// TIA Portal V18 export
FUNCTION "ST10_Auto" : Void   // FC1003, LAD
{ S7_Optimized_Access := 'FALSE' }
// stored: AutoNumber false, SetENOAutomatically false
   VAR_INPUT
      iSysMode : "RCS_SysComInterface_V1";
   END_VAR
   VAR_TEMP
      i : Int;
      tBool : Bool;
      FlankWord : Int;
   END_VAR
   VAR_TEMP   // added for the SCL form of the ladder/FBD networks
      _w1 : Bool;
      _w2 : Bool;
      _w3 : Bool;
      _w4 : Bool;
      _w5 : Bool;
      _w6 : Bool;
   END_VAR
BEGIN

REGION Network 1
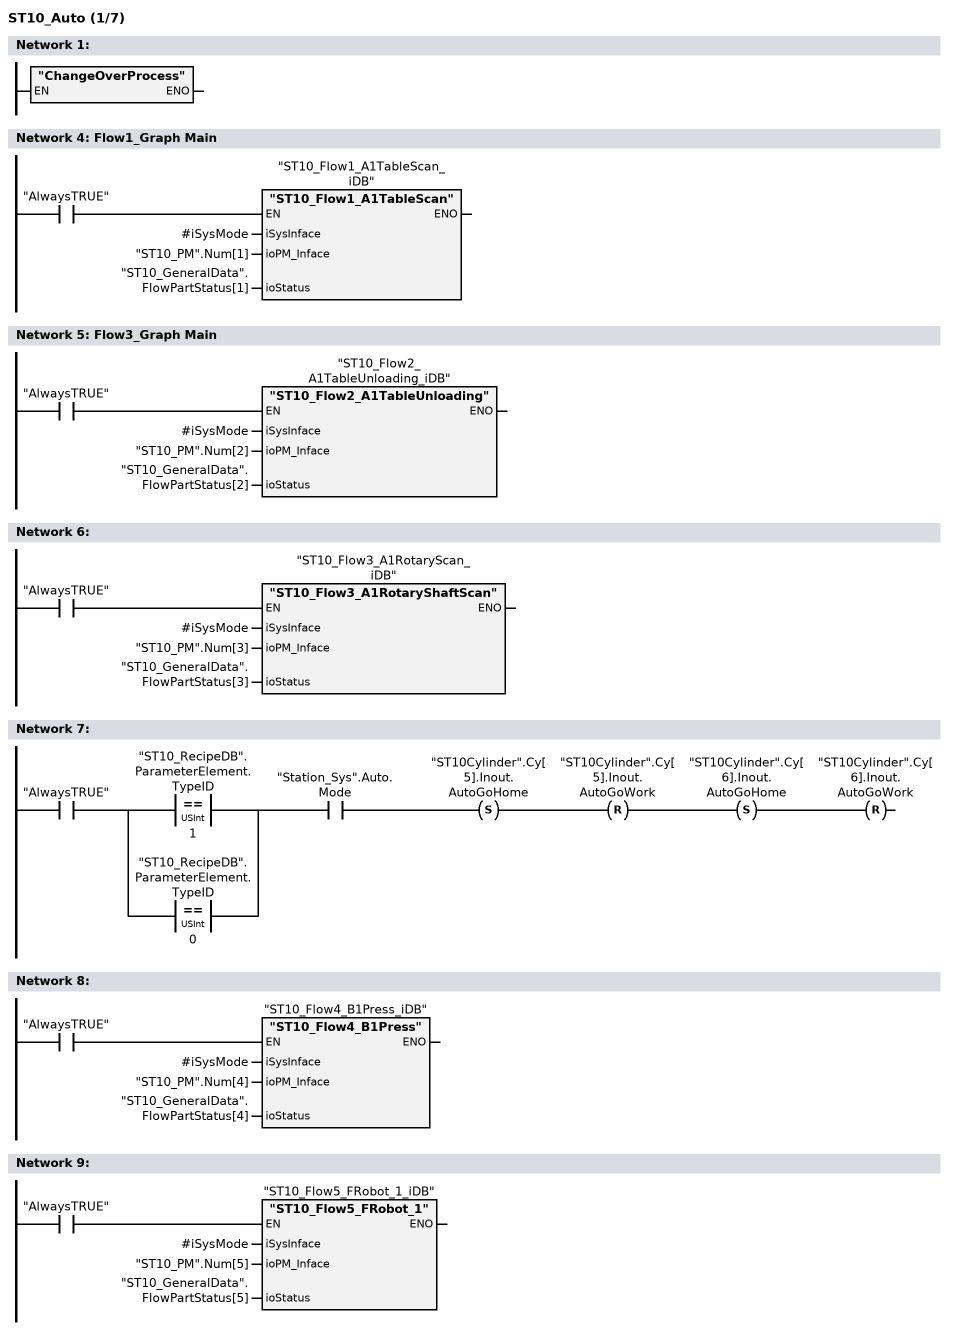
   RUNG wire#powerrail
      "ChangeOverProcess"()
   END_RUNG
   // the same network as SCL:
   "ChangeOverProcess"();
END_REGION

NETWORK
TITLE = AutoMain//自动
//Autorunning is not allowed in manual mode
      A     "Station_Sys".Manual.Mode;
      R     "Station_Sys".Auto.Running;
//one cycle interface
      A     "Station_Sys".Cmd.OneCycle;
      =     "ST10_PM".Num[1].TriggerOneCycle;
      =     "ST10_PM".Num[2].TriggerOneCycle;
      =     "ST10_PM".Num[3].TriggerOneCycle;
      =     "ST10_PM".Num[4].TriggerOneCycle;
      =     "ST10_PM".Num[5].TriggerOneCycle;
      =     "ST10_PM".Num[6].TriggerOneCycle;
      =     "ST10_PM".Num[7].TriggerOneCycle;
      =     "ST10_PM".Num[8].TriggerOneCycle;
      =     "ST10_PM".Num[11].TriggerOneCycle;
      =     "ST10_PM".Num[12].TriggerOneCycle;
      =     "ST10_PM".Num[14].TriggerOneCycle;
      =     "ST10_PM".Num[15].TriggerOneCycle;
      =     "ST10_PM".Num[16].TriggerOneCycle;
      =     "ST10_PM".Num[21].TriggerOneCycle;
      =     "ST10_PM".Num[22].TriggerOneCycle;
      =     "ST10_PM".Num[23].TriggerOneCycle;
      =     "ST10_PM".Num[24].TriggerOneCycle;


NETWORK
TITLE = InitialStatus-初始化状态
//Initilizing
      O     "ST10_PM".Num[1].InitialRun;
      O     "ST10_PM".Num[2].InitialRun;
      O     "ST10_PM".Num[3].InitialRun;
      O     "ST10_PM".Num[4].InitialRun;
      O     "ST10_PM".Num[5].InitialRun;
      O     "ST10_PM".Num[6].InitialRun;
      O     "ST10_PM".Num[7].InitialRun;
      O     "ST10_PM".Num[8].InitialRun;
      O     "ST10_PM".Num[11].InitialRun;
      O     "ST10_PM".Num[12].InitialRun;
      O     "ST10_PM".Num[14].InitialRun;
      O     "ST10_PM".Num[15].InitialRun;
      O     "ST10_PM".Num[21].InitialRun;
      O     "ST10_PM".Num[22].InitialRun;
      O     "ST10_PM".Num[23].InitialRun;
      O     "ST10_PM".Num[24].InitialRun;
      =     "Station_Sys".Initial.Running;
//Initilize ok

      A     "ST10_PM".Num[1].InitialOK;
      A     "ST10_PM".Num[2].InitialOK;
      A     "ST10_PM".Num[3].InitialOK;
      A     "ST10_PM".Num[4].InitialOK;
      A     "ST10_PM".Num[5].InitialOK;
      A     "ST10_PM".Num[6].InitialOK;
      A     "ST10_PM".Num[7].InitialOK;
      A     "ST10_PM".Num[8].InitialOK;
      A     "ST10_PM".Num[11].InitialOK;
      A     "ST10_PM".Num[12].InitialOK;
      A     "ST10_PM".Num[14].InitialOK;
      A     "ST10_PM".Num[15].InitialOK;

      A     "ST10_PM".Num[21].InitialOK;
      A     "ST10_PM".Num[22].InitialOK;
      A     "ST10_PM".Num[23].InitialOK;
      A     "ST10_PM".Num[24].InitialOK;
      =     "Station_Sys".Initial.OK;

//Auto running
      A     "Station_Sys".Auto.Mode;
      A(;
      O     "ST10_PM".Num[1].Running;
      O     "ST10_PM".Num[2].Running;
      O     "ST10_PM".Num[3].Running;
      O     "ST10_PM".Num[4].Running;
      O     "ST10_PM".Num[5].Running;
      O     "ST10_PM".Num[6].Running;
      O     "ST10_PM".Num[7].Running;
      O     "ST10_PM".Num[8].Running;
      O     "ST10_PM".Num[11].Running;
      O     "ST10_PM".Num[12].Running;
      O     "ST10_PM".Num[14].Running;
      O     "ST10_PM".Num[15].Running;

      O     "ST10_PM".Num[21].Running;
      O     "ST10_PM".Num[22].Running;
      O     "ST10_PM".Num[23].Running;
      O     "ST10_PM".Num[24].Running;
      );
// AN    "Station_Sys".Auto.AllRun
      =     "Station_Sys".Auto.Running;
//All run
      A     "ST10_PM".Num[1].Running;
      A     "ST10_PM".Num[2].Running;
      A     "ST10_PM".Num[3].Running;
      A     "ST10_PM".Num[4].Running;
      A     "ST10_PM".Num[5].Running;
      A     "ST10_PM".Num[6].Running;
      A     "ST10_PM".Num[7].Running;
      A     "ST10_PM".Num[8].Running;
      A     "ST10_PM".Num[11].Running;
      A     "ST10_PM".Num[12].Running;
      A     "ST10_PM".Num[14].Running;
      A     "ST10_PM".Num[15].Running;

      A     "ST10_PM".Num[21].Running;
      A     "ST10_PM".Num[22].Running;
      A     "ST10_PM".Num[23].Running;
      A     "ST10_PM".Num[24].Running;
      =     "Station_Sys".Auto.AllRun;




REGION Network 4: Flow1_Graph Main
   RUNG wire#powerrail
      Contact( "AlwaysTRUE" )
      "ST10_Flow1_A1TableScan_iDB"(iSysInface := #iSysMode, ioPM_Inface := "ST10_PM".Num[1], ioStatus := "ST10_GeneralData".FlowPartStatus[1])
   END_RUNG
   // the same network as SCL:
   IF "AlwaysTRUE" THEN
       "ST10_Flow1_A1TableScan_iDB"(iSysInface := #iSysMode,   // "ST10_Flow1_A1TableScan"
                               ioPM_Inface := "ST10_PM".Num[1],
                               ioStatus := "ST10_GeneralData".FlowPartStatus[1]);
   END_IF;
END_REGION

REGION Network 5: Flow3_Graph Main
   RUNG wire#powerrail
      Contact( "AlwaysTRUE" )
      "ST10_Flow2_A1TableUnloading_iDB"(iSysInface := #iSysMode, ioPM_Inface := "ST10_PM".Num[2], ioStatus := "ST10_GeneralData".FlowPartStatus[2])
   END_RUNG
   // the same network as SCL:
   IF "AlwaysTRUE" THEN
       "ST10_Flow2_A1TableUnloading_iDB"(iSysInface := #iSysMode,   // "ST10_Flow2_A1TableUnloading"
                               ioPM_Inface := "ST10_PM".Num[2],
                               ioStatus := "ST10_GeneralData".FlowPartStatus[2]);
   END_IF;
END_REGION

REGION Network 6
   RUNG wire#powerrail
      Contact( "AlwaysTRUE" )
      "ST10_Flow3_A1RotaryScan_iDB"(iSysInface := #iSysMode, ioPM_Inface := "ST10_PM".Num[3], ioStatus := "ST10_GeneralData".FlowPartStatus[3])
   END_RUNG
   // the same network as SCL:
   IF "AlwaysTRUE" THEN
       "ST10_Flow3_A1RotaryScan_iDB"(iSysInface := #iSysMode,   // "ST10_Flow3_A1RotaryShaftScan"
                               ioPM_Inface := "ST10_PM".Num[3],
                               ioStatus := "ST10_GeneralData".FlowPartStatus[3]);
   END_IF;
END_REGION

REGION Network 7
   RUNG wire#powerrail
      Contact( "AlwaysTRUE" )
      wire#w1
      { S7_Templates := "SrcType := USInt" } EQ_Contact(in1 := "ST10_RecipeDB".ParameterElement.TypeID, in2 := 1)
      wire#w2
      Contact( "Station_Sys".Auto.Mode )
      S_Coil( "ST10Cylinder".Cy[5].Inout.AutoGoHome )
      R_Coil( "ST10Cylinder".Cy[5].Inout.AutoGoWork )
      S_Coil( "ST10Cylinder".Cy[6].Inout.AutoGoHome )
      R_Coil( "ST10Cylinder".Cy[6].Inout.AutoGoWork )
   END_RUNG
   RUNG wire#w1
      { S7_Templates := "SrcType := USInt" } EQ_Contact(in1 := "ST10_RecipeDB".ParameterElement.TypeID, in2 := 0)
   END_RUNG wire#w2
   // the same network as SCL:
   IF "AlwaysTRUE" AND (("ST10_RecipeDB".ParameterElement.TypeID = 1) OR ("ST10_RecipeDB".ParameterElement.TypeID = 0)) AND "Station_Sys".Auto.Mode THEN
       "ST10Cylinder".Cy[5].Inout.AutoGoHome := TRUE;
       "ST10Cylinder".Cy[5].Inout.AutoGoWork := FALSE;
       "ST10Cylinder".Cy[6].Inout.AutoGoHome := TRUE;
       "ST10Cylinder".Cy[6].Inout.AutoGoWork := FALSE;
   END_IF;
END_REGION

REGION Network 8
   RUNG wire#powerrail
      Contact( "AlwaysTRUE" )
      "ST10_Flow4_B1Press_iDB"(iSysInface := #iSysMode, ioPM_Inface := "ST10_PM".Num[4], ioStatus := "ST10_GeneralData".FlowPartStatus[4])
   END_RUNG
   // the same network as SCL:
   IF "AlwaysTRUE" THEN
       "ST10_Flow4_B1Press_iDB"(iSysInface := #iSysMode,   // "ST10_Flow4_B1Press"
                               ioPM_Inface := "ST10_PM".Num[4],
                               ioStatus := "ST10_GeneralData".FlowPartStatus[4]);
   END_IF;
END_REGION

REGION Network 9
   RUNG wire#powerrail
      Contact( "AlwaysTRUE" )
      "ST10_Flow5_FRobot_1_iDB"(iSysInface := #iSysMode, ioPM_Inface := "ST10_PM".Num[5], ioStatus := "ST10_GeneralData".FlowPartStatus[5])
   END_RUNG
   // the same network as SCL:
   IF "AlwaysTRUE" THEN
       "ST10_Flow5_FRobot_1_iDB"(iSysInface := #iSysMode,   // "ST10_Flow5_FRobot_1"
                               ioPM_Inface := "ST10_PM".Num[5],
                               ioStatus := "ST10_GeneralData".FlowPartStatus[5]);
   END_IF;
END_REGION

REGION Network 10
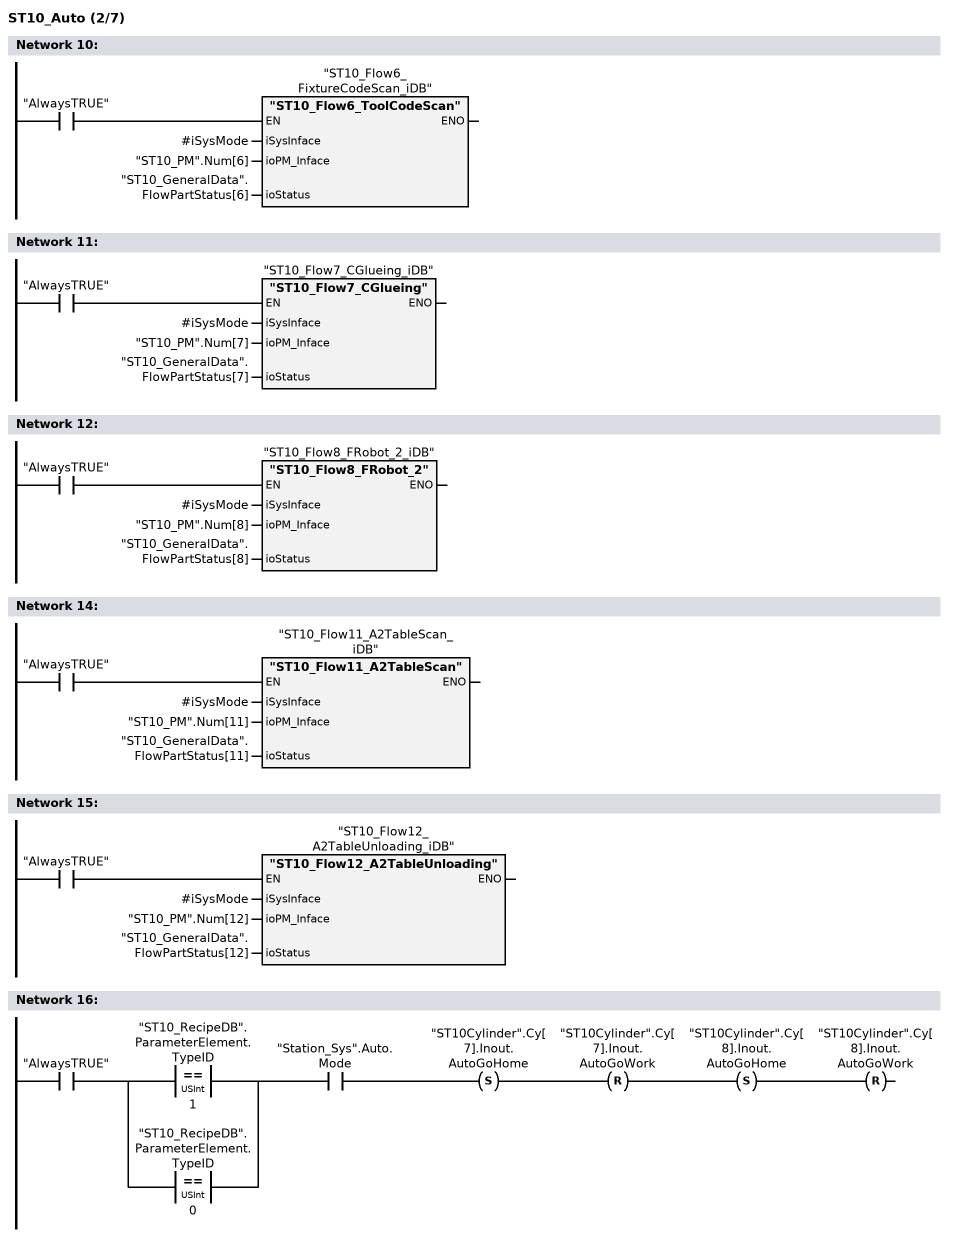
   RUNG wire#powerrail
      Contact( "AlwaysTRUE" )
      "ST10_Flow6_FixtureCodeScan_iDB"(iSysInface := #iSysMode, ioPM_Inface := "ST10_PM".Num[6], ioStatus := "ST10_GeneralData".FlowPartStatus[6])
   END_RUNG
   // the same network as SCL:
   IF "AlwaysTRUE" THEN
       "ST10_Flow6_FixtureCodeScan_iDB"(iSysInface := #iSysMode,   // "ST10_Flow6_ToolCodeScan"
                               ioPM_Inface := "ST10_PM".Num[6],
                               ioStatus := "ST10_GeneralData".FlowPartStatus[6]);
   END_IF;
END_REGION

REGION Network 11
   RUNG wire#powerrail
      Contact( "AlwaysTRUE" )
      "ST10_Flow7_CGlueing_iDB"(iSysInface := #iSysMode, ioPM_Inface := "ST10_PM".Num[7], ioStatus := "ST10_GeneralData".FlowPartStatus[7])
   END_RUNG
   // the same network as SCL:
   IF "AlwaysTRUE" THEN
       "ST10_Flow7_CGlueing_iDB"(iSysInface := #iSysMode,   // "ST10_Flow7_CGlueing"
                               ioPM_Inface := "ST10_PM".Num[7],
                               ioStatus := "ST10_GeneralData".FlowPartStatus[7]);
   END_IF;
END_REGION

REGION Network 12
   RUNG wire#powerrail
      Contact( "AlwaysTRUE" )
      "ST10_Flow8_FRobot_2_iDB"(iSysInface := #iSysMode, ioPM_Inface := "ST10_PM".Num[8], ioStatus := "ST10_GeneralData".FlowPartStatus[8])
   END_RUNG
   // the same network as SCL:
   IF "AlwaysTRUE" THEN
       "ST10_Flow8_FRobot_2_iDB"(iSysInface := #iSysMode,   // "ST10_Flow8_FRobot_2"
                               ioPM_Inface := "ST10_PM".Num[8],
                               ioStatus := "ST10_GeneralData".FlowPartStatus[8]);
   END_IF;
END_REGION

REGION Network 14
   RUNG wire#powerrail
      Contact( "AlwaysTRUE" )
      "ST10_Flow11_A2TableScan_iDB"(iSysInface := #iSysMode, ioPM_Inface := "ST10_PM".Num[11], ioStatus := "ST10_GeneralData".FlowPartStatus[11])
   END_RUNG
   // the same network as SCL:
   IF "AlwaysTRUE" THEN
       "ST10_Flow11_A2TableScan_iDB"(iSysInface := #iSysMode,   // "ST10_Flow11_A2TableScan"
                               ioPM_Inface := "ST10_PM".Num[11],
                               ioStatus := "ST10_GeneralData".FlowPartStatus[11]);
   END_IF;
END_REGION

REGION Network 15
   RUNG wire#powerrail
      Contact( "AlwaysTRUE" )
      "ST10_Flow12_A2TableUnloading_iDB"(iSysInface := #iSysMode, ioPM_Inface := "ST10_PM".Num[12], ioStatus := "ST10_GeneralData".FlowPartStatus[12])
   END_RUNG
   // the same network as SCL:
   IF "AlwaysTRUE" THEN
       "ST10_Flow12_A2TableUnloading_iDB"(iSysInface := #iSysMode,   // "ST10_Flow12_A2TableUnloading"
                               ioPM_Inface := "ST10_PM".Num[12],
                               ioStatus := "ST10_GeneralData".FlowPartStatus[12]);
   END_IF;
END_REGION

REGION Network 16
   RUNG wire#powerrail
      Contact( "AlwaysTRUE" )
      wire#w1
      { S7_Templates := "SrcType := USInt" } EQ_Contact(in1 := "ST10_RecipeDB".ParameterElement.TypeID, in2 := 1)
      wire#w2
      Contact( "Station_Sys".Auto.Mode )
      S_Coil( "ST10Cylinder".Cy[7].Inout.AutoGoHome )
      R_Coil( "ST10Cylinder".Cy[7].Inout.AutoGoWork )
      S_Coil( "ST10Cylinder".Cy[8].Inout.AutoGoHome )
      R_Coil( "ST10Cylinder".Cy[8].Inout.AutoGoWork )
   END_RUNG
   RUNG wire#w1
      { S7_Templates := "SrcType := USInt" } EQ_Contact(in1 := "ST10_RecipeDB".ParameterElement.TypeID, in2 := 0)
   END_RUNG wire#w2
   // the same network as SCL:
   IF "AlwaysTRUE" AND (("ST10_RecipeDB".ParameterElement.TypeID = 1) OR ("ST10_RecipeDB".ParameterElement.TypeID = 0)) AND "Station_Sys".Auto.Mode THEN
       "ST10Cylinder".Cy[7].Inout.AutoGoHome := TRUE;
       "ST10Cylinder".Cy[7].Inout.AutoGoWork := FALSE;
       "ST10Cylinder".Cy[8].Inout.AutoGoHome := TRUE;
       "ST10Cylinder".Cy[8].Inout.AutoGoWork := FALSE;
   END_IF;
END_REGION

REGION Network 17
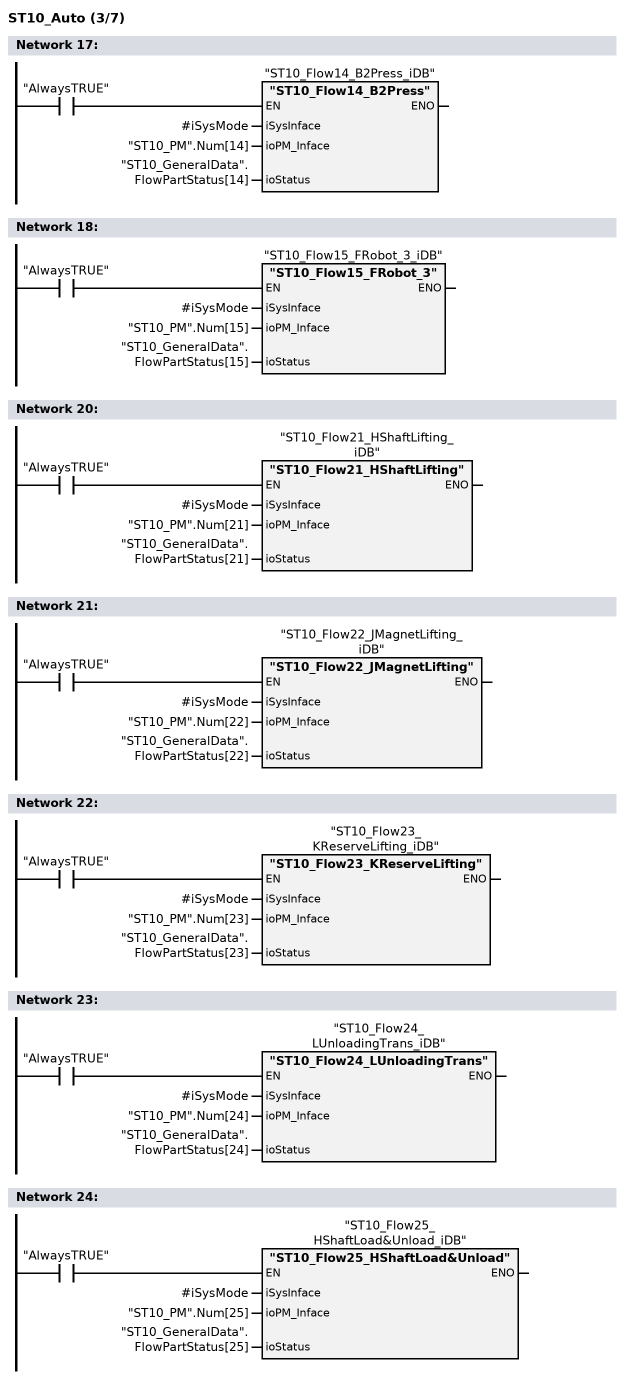
   RUNG wire#powerrail
      Contact( "AlwaysTRUE" )
      "ST10_Flow14_B2Press_iDB"(iSysInface := #iSysMode, ioPM_Inface := "ST10_PM".Num[14], ioStatus := "ST10_GeneralData".FlowPartStatus[14])
   END_RUNG
   // the same network as SCL:
   IF "AlwaysTRUE" THEN
       "ST10_Flow14_B2Press_iDB"(iSysInface := #iSysMode,   // "ST10_Flow14_B2Press"
                               ioPM_Inface := "ST10_PM".Num[14],
                               ioStatus := "ST10_GeneralData".FlowPartStatus[14]);
   END_IF;
END_REGION

REGION Network 18
   RUNG wire#powerrail
      Contact( "AlwaysTRUE" )
      "ST10_Flow15_FRobot_3_iDB"(iSysInface := #iSysMode, ioPM_Inface := "ST10_PM".Num[15], ioStatus := "ST10_GeneralData".FlowPartStatus[15])
   END_RUNG
   // the same network as SCL:
   IF "AlwaysTRUE" THEN
       "ST10_Flow15_FRobot_3_iDB"(iSysInface := #iSysMode,   // "ST10_Flow15_FRobot_3"
                               ioPM_Inface := "ST10_PM".Num[15],
                               ioStatus := "ST10_GeneralData".FlowPartStatus[15]);
   END_IF;
END_REGION

REGION Network 20
   RUNG wire#powerrail
      Contact( "AlwaysTRUE" )
      "ST10_Flow21_HShaftLifting_iDB"(iSysInface := #iSysMode, ioPM_Inface := "ST10_PM".Num[21], ioStatus := "ST10_GeneralData".FlowPartStatus[21])
   END_RUNG
   // the same network as SCL:
   IF "AlwaysTRUE" THEN
       "ST10_Flow21_HShaftLifting_iDB"(iSysInface := #iSysMode,   // "ST10_Flow21_HShaftLifting"
                               ioPM_Inface := "ST10_PM".Num[21],
                               ioStatus := "ST10_GeneralData".FlowPartStatus[21]);
   END_IF;
END_REGION

REGION Network 21
   RUNG wire#powerrail
      Contact( "AlwaysTRUE" )
      "ST10_Flow22_JMagnetLifting_iDB"(iSysInface := #iSysMode, ioPM_Inface := "ST10_PM".Num[22], ioStatus := "ST10_GeneralData".FlowPartStatus[22])
   END_RUNG
   // the same network as SCL:
   IF "AlwaysTRUE" THEN
       "ST10_Flow22_JMagnetLifting_iDB"(iSysInface := #iSysMode,   // "ST10_Flow22_JMagnetLifting"
                               ioPM_Inface := "ST10_PM".Num[22],
                               ioStatus := "ST10_GeneralData".FlowPartStatus[22]);
   END_IF;
END_REGION

REGION Network 22
   RUNG wire#powerrail
      Contact( "AlwaysTRUE" )
      "ST10_Flow23_KReserveLifting_iDB"(iSysInface := #iSysMode, ioPM_Inface := "ST10_PM".Num[23], ioStatus := "ST10_GeneralData".FlowPartStatus[23])
   END_RUNG
   // the same network as SCL:
   IF "AlwaysTRUE" THEN
       "ST10_Flow23_KReserveLifting_iDB"(iSysInface := #iSysMode,   // "ST10_Flow23_KReserveLifting"
                               ioPM_Inface := "ST10_PM".Num[23],
                               ioStatus := "ST10_GeneralData".FlowPartStatus[23]);
   END_IF;
END_REGION

REGION Network 23
   RUNG wire#powerrail
      Contact( "AlwaysTRUE" )
      "ST10_Flow24_LUnloadingTrans_iDB"(iSysInface := #iSysMode, ioPM_Inface := "ST10_PM".Num[24], ioStatus := "ST10_GeneralData".FlowPartStatus[24])
   END_RUNG
   // the same network as SCL:
   IF "AlwaysTRUE" THEN
       "ST10_Flow24_LUnloadingTrans_iDB"(iSysInface := #iSysMode,   // "ST10_Flow24_LUnloadingTrans"
                               ioPM_Inface := "ST10_PM".Num[24],
                               ioStatus := "ST10_GeneralData".FlowPartStatus[24]);
   END_IF;
END_REGION

REGION Network 24
   RUNG wire#powerrail
      Contact( "AlwaysTRUE" )
      "ST10_Flow25_HShaftLoad&Unload_iDB"(iSysInface := #iSysMode, ioPM_Inface := "ST10_PM".Num[25], ioStatus := "ST10_GeneralData".FlowPartStatus[25])
   END_RUNG
   // the same network as SCL:
   IF "AlwaysTRUE" THEN
       "ST10_Flow25_HShaftLoad&Unload_iDB"(iSysInface := #iSysMode,   // "ST10_Flow25_HShaftLoad&Unload"
                               ioPM_Inface := "ST10_PM".Num[25],
                               ioStatus := "ST10_GeneralData".FlowPartStatus[25]);
   END_IF;
END_REGION

REGION Network 25
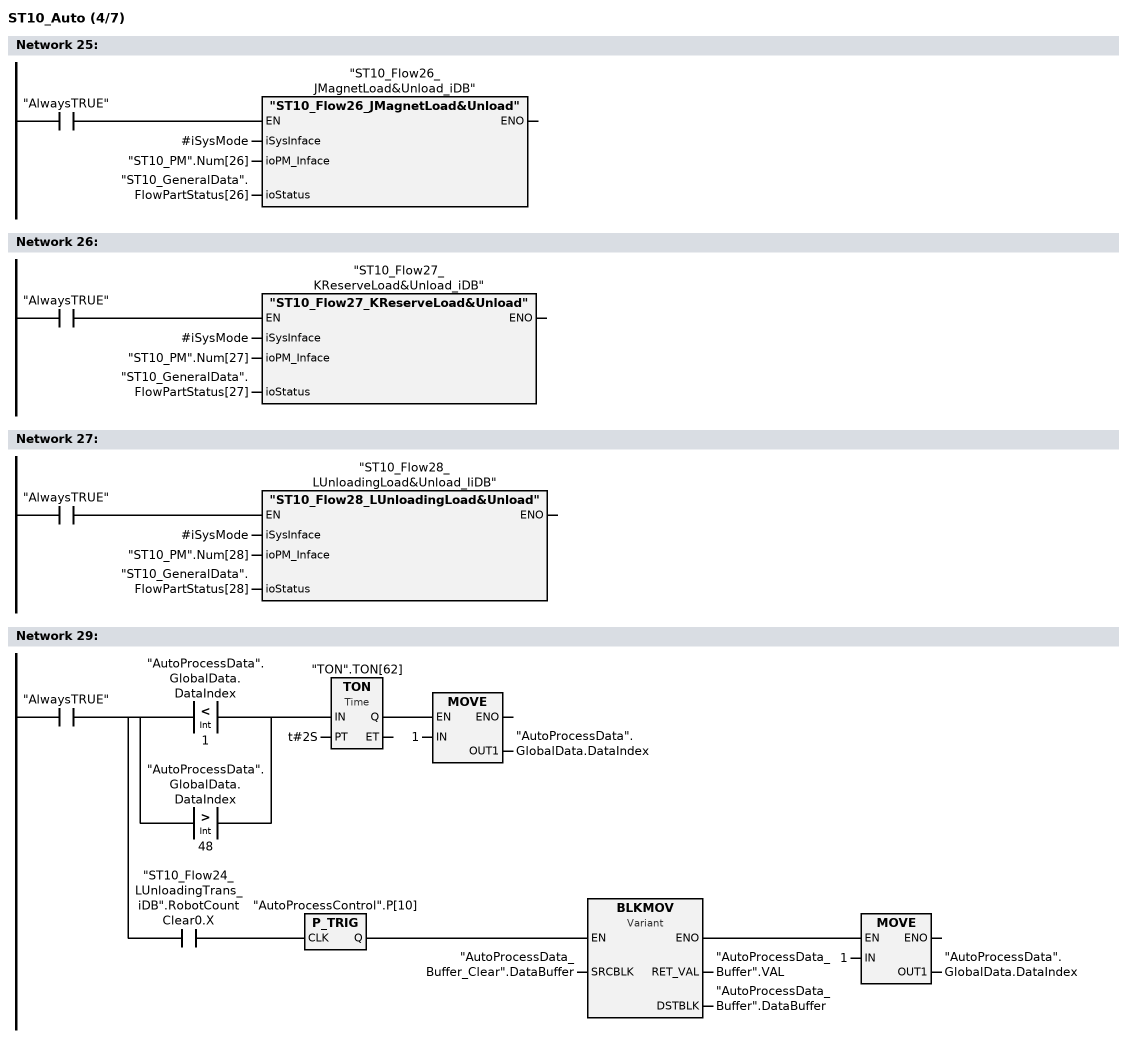
   RUNG wire#powerrail
      Contact( "AlwaysTRUE" )
      "ST10_Flow26_JMagnetLoad&Unload_iDB"(iSysInface := #iSysMode, ioPM_Inface := "ST10_PM".Num[26], ioStatus := "ST10_GeneralData".FlowPartStatus[26])
   END_RUNG
   // the same network as SCL:
   IF "AlwaysTRUE" THEN
       "ST10_Flow26_JMagnetLoad&Unload_iDB"(iSysInface := #iSysMode,   // "ST10_Flow26_JMagnetLoad&Unload"
                               ioPM_Inface := "ST10_PM".Num[26],
                               ioStatus := "ST10_GeneralData".FlowPartStatus[26]);
   END_IF;
END_REGION

REGION Network 26
   RUNG wire#powerrail
      Contact( "AlwaysTRUE" )
      "ST10_Flow27_KReserveLoad&Unload_iDB"(iSysInface := #iSysMode, ioPM_Inface := "ST10_PM".Num[27], ioStatus := "ST10_GeneralData".FlowPartStatus[27])
   END_RUNG
   // the same network as SCL:
   IF "AlwaysTRUE" THEN
       "ST10_Flow27_KReserveLoad&Unload_iDB"(iSysInface := #iSysMode,   // "ST10_Flow27_KReserveLoad&Unload"
                               ioPM_Inface := "ST10_PM".Num[27],
                               ioStatus := "ST10_GeneralData".FlowPartStatus[27]);
   END_IF;
END_REGION

REGION Network 27
   RUNG wire#powerrail
      Contact( "AlwaysTRUE" )
      "ST10_Flow28_LUnloadingLoad&Unload_IiDB"(iSysInface := #iSysMode, ioPM_Inface := "ST10_PM".Num[28], ioStatus := "ST10_GeneralData".FlowPartStatus[28])
   END_RUNG
   // the same network as SCL:
   IF "AlwaysTRUE" THEN
       "ST10_Flow28_LUnloadingLoad&Unload_IiDB"(iSysInface := #iSysMode,   // "ST10_Flow28_LUnloadingLoad&Unload"
                               ioPM_Inface := "ST10_PM".Num[28],
                               ioStatus := "ST10_GeneralData".FlowPartStatus[28]);
   END_IF;
END_REGION

REGION Network 29
   RUNG wire#powerrail
      Contact( "AlwaysTRUE" )
      wire#w1
      { S7_Templates := "SrcType := Int" } LT_Contact(in1 := "AutoProcessData".GlobalData.DataIndex, in2 := 1)
      wire#w2
      { S7_Templates := "time_type := Time" } "TON".TON[62].TON(pt := t#2S, et =>)
      Move(in := 1, out1 => "AutoProcessData".GlobalData.DataIndex)
   END_RUNG
   RUNG wire#w1
      { S7_Templates := "SrcType := Int" } GT_Contact(in1 := "AutoProcessData".GlobalData.DataIndex, in2 := 48)
   END_RUNG wire#w2
   RUNG wire#w1
      Contact( "ST10_Flow24_LUnloadingTrans_iDB".RobotCountClear0.X )
      P_Trig( "AutoProcessControl".P[10] )
      { S7_Templates := "blk_type := Variant" } BLKMOV(SRCBLK := "AutoProcessData_Buffer_Clear".DataBuffer, RET_VAL => "AutoProcessData_Buffer".VAL, DSTBLK => "AutoProcessData_Buffer".DataBuffer)
      Move(in := 1, out1 => "AutoProcessData".GlobalData.DataIndex)
   END_RUNG
   // the same network as SCL:
   "TON".TON[62].TON(IN := "AlwaysTRUE" AND (("AutoProcessData".GlobalData.DataIndex < 1) OR ("AutoProcessData".GlobalData.DataIndex > 48)),
                     PT := t#2S);
   IF "TON".TON[62].Q THEN "AutoProcessData".GlobalData.DataIndex := 1; END_IF;
   #_w1 := "AlwaysTRUE" AND "ST10_Flow24_LUnloadingTrans_iDB".RobotCountClear0.X;
   #_w2 := #_w1 AND NOT "AutoProcessControl".P[10];   // rising edge
   "AutoProcessControl".P[10] := #_w1;
   "AutoProcessData_Buffer".VAL := BLKMOV(EN := #_w2,
                           SRCBLK := "AutoProcessData_Buffer_Clear".DataBuffer,
                           DSTBLK => "AutoProcessData_Buffer".DataBuffer,
                           ENO => #_w3);
   IF #_w3 THEN "AutoProcessData".GlobalData.DataIndex := 1; END_IF;
END_REGION

REGION Network 30
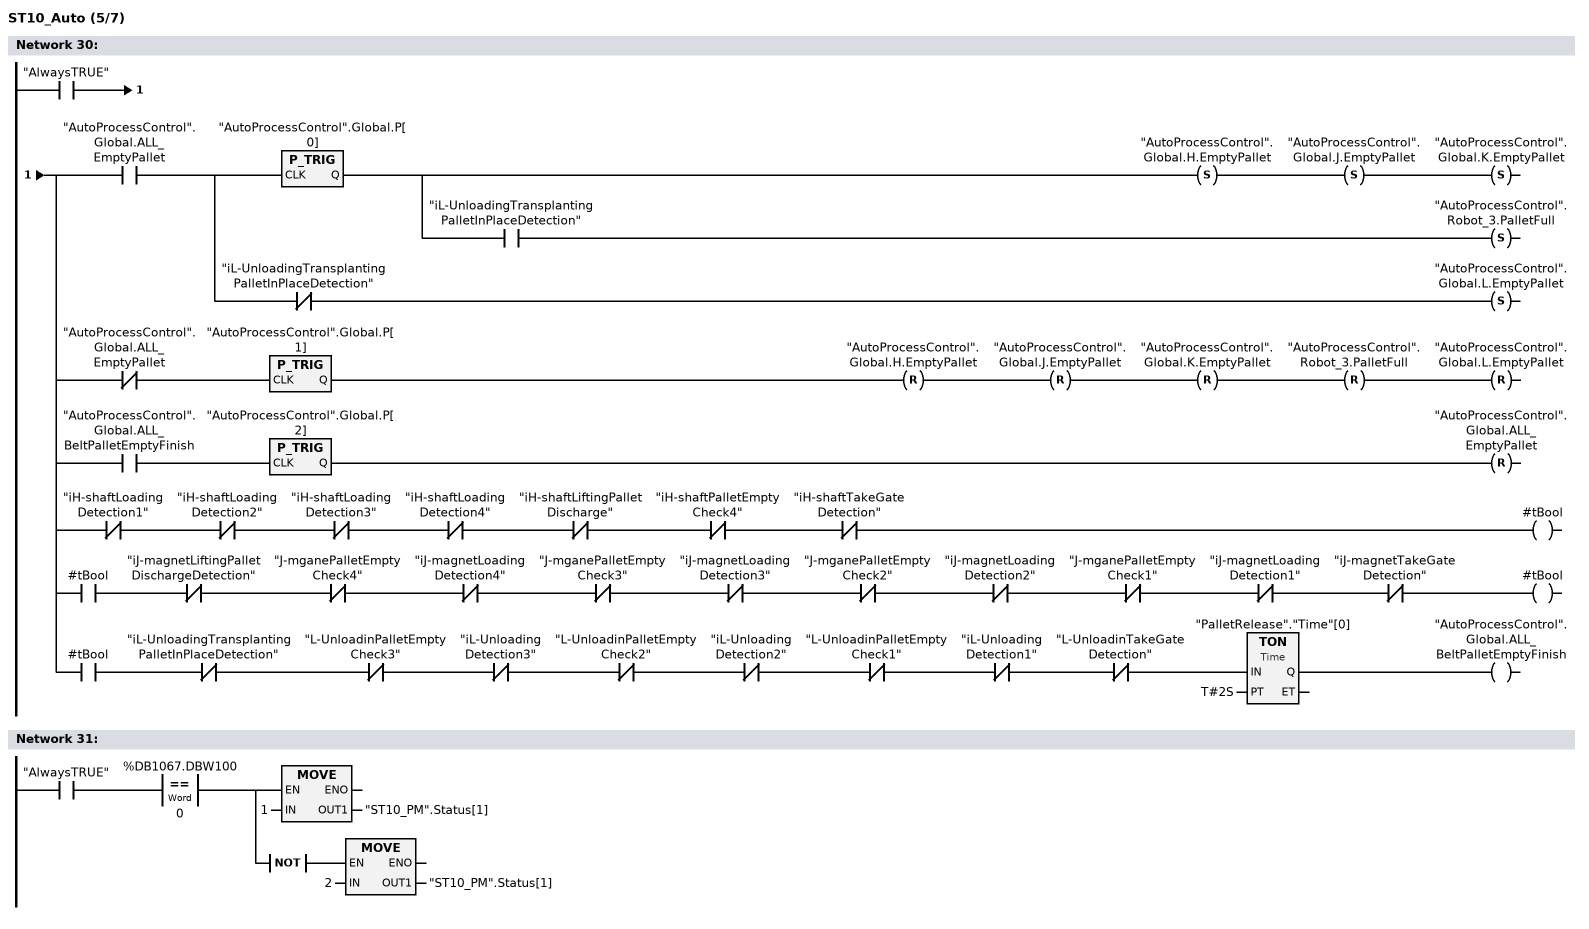
   RUNG wire#powerrail
      Contact( "AlwaysTRUE" )
      wire#w1
      Contact( "AutoProcessControl".Global.ALL_EmptyPallet )
      wire#w2
      P_Trig( "AutoProcessControl".Global.P[0] )
      wire#w3
      S_Coil( "AutoProcessControl".Global.H.EmptyPallet )
      S_Coil( "AutoProcessControl".Global.J.EmptyPallet )
      S_Coil( "AutoProcessControl".Global.K.EmptyPallet )
   END_RUNG
   RUNG wire#w3
      Contact( "iL-UnloadingTransplantingPalletInPlaceDetection" )
      S_Coil( "AutoProcessControl".Robot_3.PalletFull )
   END_RUNG
   RUNG wire#w2
      I_Contact( "iL-UnloadingTransplantingPalletInPlaceDetection" )
      S_Coil( "AutoProcessControl".Global.L.EmptyPallet )
   END_RUNG
   RUNG wire#w1
      I_Contact( "AutoProcessControl".Global.ALL_EmptyPallet )
      P_Trig( "AutoProcessControl".Global.P[1] )
      R_Coil( "AutoProcessControl".Global.H.EmptyPallet )
      R_Coil( "AutoProcessControl".Global.J.EmptyPallet )
      R_Coil( "AutoProcessControl".Global.K.EmptyPallet )
      R_Coil( "AutoProcessControl".Robot_3.PalletFull )
      R_Coil( "AutoProcessControl".Global.L.EmptyPallet )
   END_RUNG
   RUNG wire#w1
      Contact( "AutoProcessControl".Global.ALL_BeltPalletEmptyFinish )
      P_Trig( "AutoProcessControl".Global.P[2] )
      R_Coil( "AutoProcessControl".Global.ALL_EmptyPallet )
   END_RUNG
   RUNG wire#w1
      I_Contact( "iH-shaftLoadingDetection1" )
      I_Contact( "iH-shaftLoadingDetection2" )
      I_Contact( "iH-shaftLoadingDetection3" )
      I_Contact( "iH-shaftLoadingDetection4" )
      I_Contact( "iH-shaftLiftingPalletDischarge" )
      I_Contact( "iH-shaftPalletEmptyCheck4" )
      I_Contact( "iH-shaftTakeGateDetection" )
      Coil( #tBool )
   END_RUNG
   RUNG wire#w1
      Contact( #tBool )
      I_Contact( "iJ-magnetLiftingPalletDischargeDetection" )
      I_Contact( "J-mganePalletEmptyCheck4" )
      I_Contact( "iJ-magnetLoadingDetection4" )
      I_Contact( "J-mganePalletEmptyCheck3" )
      I_Contact( "iJ-magnetLoadingDetection3" )
      I_Contact( "J-mganePalletEmptyCheck2" )
      I_Contact( "iJ-magnetLoadingDetection2" )
      I_Contact( "J-mganePalletEmptyCheck1" )
      I_Contact( "iJ-magnetLoadingDetection1" )
      I_Contact( "iJ-magnetTakeGateDetection" )
      Coil( #tBool )
   END_RUNG
   RUNG wire#w1
      Contact( #tBool )
      I_Contact( "iL-UnloadingTransplantingPalletInPlaceDetection" )
      I_Contact( "L-UnloadinPalletEmptyCheck3" )
      I_Contact( "iL-UnloadingDetection3" )
      I_Contact( "L-UnloadinPalletEmptyCheck2" )
      I_Contact( "iL-UnloadingDetection2" )
      I_Contact( "L-UnloadinPalletEmptyCheck1" )
      I_Contact( "iL-UnloadingDetection1" )
      I_Contact( "L-UnloadinTakeGateDetection" )
      { S7_Templates := "time_type := Time" } "PalletRelease"."Time"[0].TON(pt := T#2S, et =>)
      Coil( "AutoProcessControl".Global.ALL_BeltPalletEmptyFinish )
   END_RUNG
   // the same network as SCL:
   #_w1 := "AlwaysTRUE" AND "AutoProcessControl".Global.ALL_EmptyPallet;
   #_w2 := #_w1 AND NOT "AutoProcessControl".Global.P[0];   // rising edge
   "AutoProcessControl".Global.P[0] := #_w1;
   IF #_w2 THEN
       "AutoProcessControl".Global.H.EmptyPallet := TRUE;
       "AutoProcessControl".Global.J.EmptyPallet := TRUE;
       "AutoProcessControl".Global.K.EmptyPallet := TRUE;
   END_IF;
   IF #_w2 AND "iL-UnloadingTransplantingPalletInPlaceDetection" THEN
       "AutoProcessControl".Robot_3.PalletFull := TRUE;
   END_IF;
   IF #_w1 AND NOT "iL-UnloadingTransplantingPalletInPlaceDetection" THEN
       "AutoProcessControl".Global.L.EmptyPallet := TRUE;
   END_IF;
   #_w3 := "AlwaysTRUE" AND NOT "AutoProcessControl".Global.ALL_EmptyPallet;
   #_w4 := #_w3 AND NOT "AutoProcessControl".Global.P[1];   // rising edge
   "AutoProcessControl".Global.P[1] := #_w3;
   IF #_w4 THEN
       "AutoProcessControl".Global.H.EmptyPallet := FALSE;
       "AutoProcessControl".Global.J.EmptyPallet := FALSE;
       "AutoProcessControl".Global.K.EmptyPallet := FALSE;
       "AutoProcessControl".Robot_3.PalletFull := FALSE;
       "AutoProcessControl".Global.L.EmptyPallet := FALSE;
   END_IF;
   #_w5 := "AlwaysTRUE" AND "AutoProcessControl".Global.ALL_BeltPalletEmptyFinish;
   #_w6 := #_w5 AND NOT "AutoProcessControl".Global.P[2];   // rising edge
   "AutoProcessControl".Global.P[2] := #_w5;
   IF #_w6 THEN "AutoProcessControl".Global.ALL_EmptyPallet := FALSE; END_IF;
   #tBool := "AlwaysTRUE" AND NOT "iH-shaftLoadingDetection1" AND NOT "iH-shaftLoadingDetection2" AND NOT "iH-shaftLoadingDetection3" AND NOT "iH-shaftLoadingDetection4" AND NOT "iH-shaftLiftingPalletDischarge" AND NOT "iH-shaftPalletEmptyCheck4" AND NOT "iH-shaftTakeGateDetection";
   #tBool := "AlwaysTRUE" AND #tBool AND NOT "iJ-magnetLiftingPalletDischargeDetection" AND NOT "J-mganePalletEmptyCheck4" AND NOT "iJ-magnetLoadingDetection4" AND NOT "J-mganePalletEmptyCheck3" AND NOT "iJ-magnetLoadingDetection3" AND NOT "J-mganePalletEmptyCheck2" AND NOT "iJ-magnetLoadingDetection2" AND NOT "J-mganePalletEmptyCheck1" AND NOT "iJ-magnetLoadingDetection1" AND NOT "iJ-magnetTakeGateDetection";
   "PalletRelease"."Time"[0].TON(IN := "AlwaysTRUE" AND #tBool AND NOT "iL-UnloadingTransplantingPalletInPlaceDetection" AND NOT "L-UnloadinPalletEmptyCheck3" AND NOT "iL-UnloadingDetection3" AND NOT "L-UnloadinPalletEmptyCheck2" AND NOT "iL-UnloadingDetection2" AND NOT "L-UnloadinPalletEmptyCheck1" AND NOT "iL-UnloadingDetection1" AND NOT "L-UnloadinTakeGateDetection",
                           PT := T#2S);
   "AutoProcessControl".Global.ALL_BeltPalletEmptyFinish := "PalletRelease"."Time"[0].Q;
END_REGION

REGION Network 31
   RUNG wire#powerrail
      Contact( "AlwaysTRUE" )
      { S7_Templates := "SrcType := Word" } EQ_Contact(in1 := %DB1067.DBW100, in2 := 0)
      wire#w1
      Move(in := 1, out1 => "ST10_PM".Status[1])
   END_RUNG
   RUNG wire#w1
      Not()
      Move(in := 2, out1 => "ST10_PM".Status[1])
   END_RUNG
   // the same network as SCL:
   #_w1 := "AlwaysTRUE" AND (%DB1067.DBW100 = 0);
   IF #_w1 THEN "ST10_PM".Status[1] := 1; END_IF;
   IF NOT #_w1 THEN "ST10_PM".Status[1] := 2; END_IF;
END_REGION

REGION Network 33
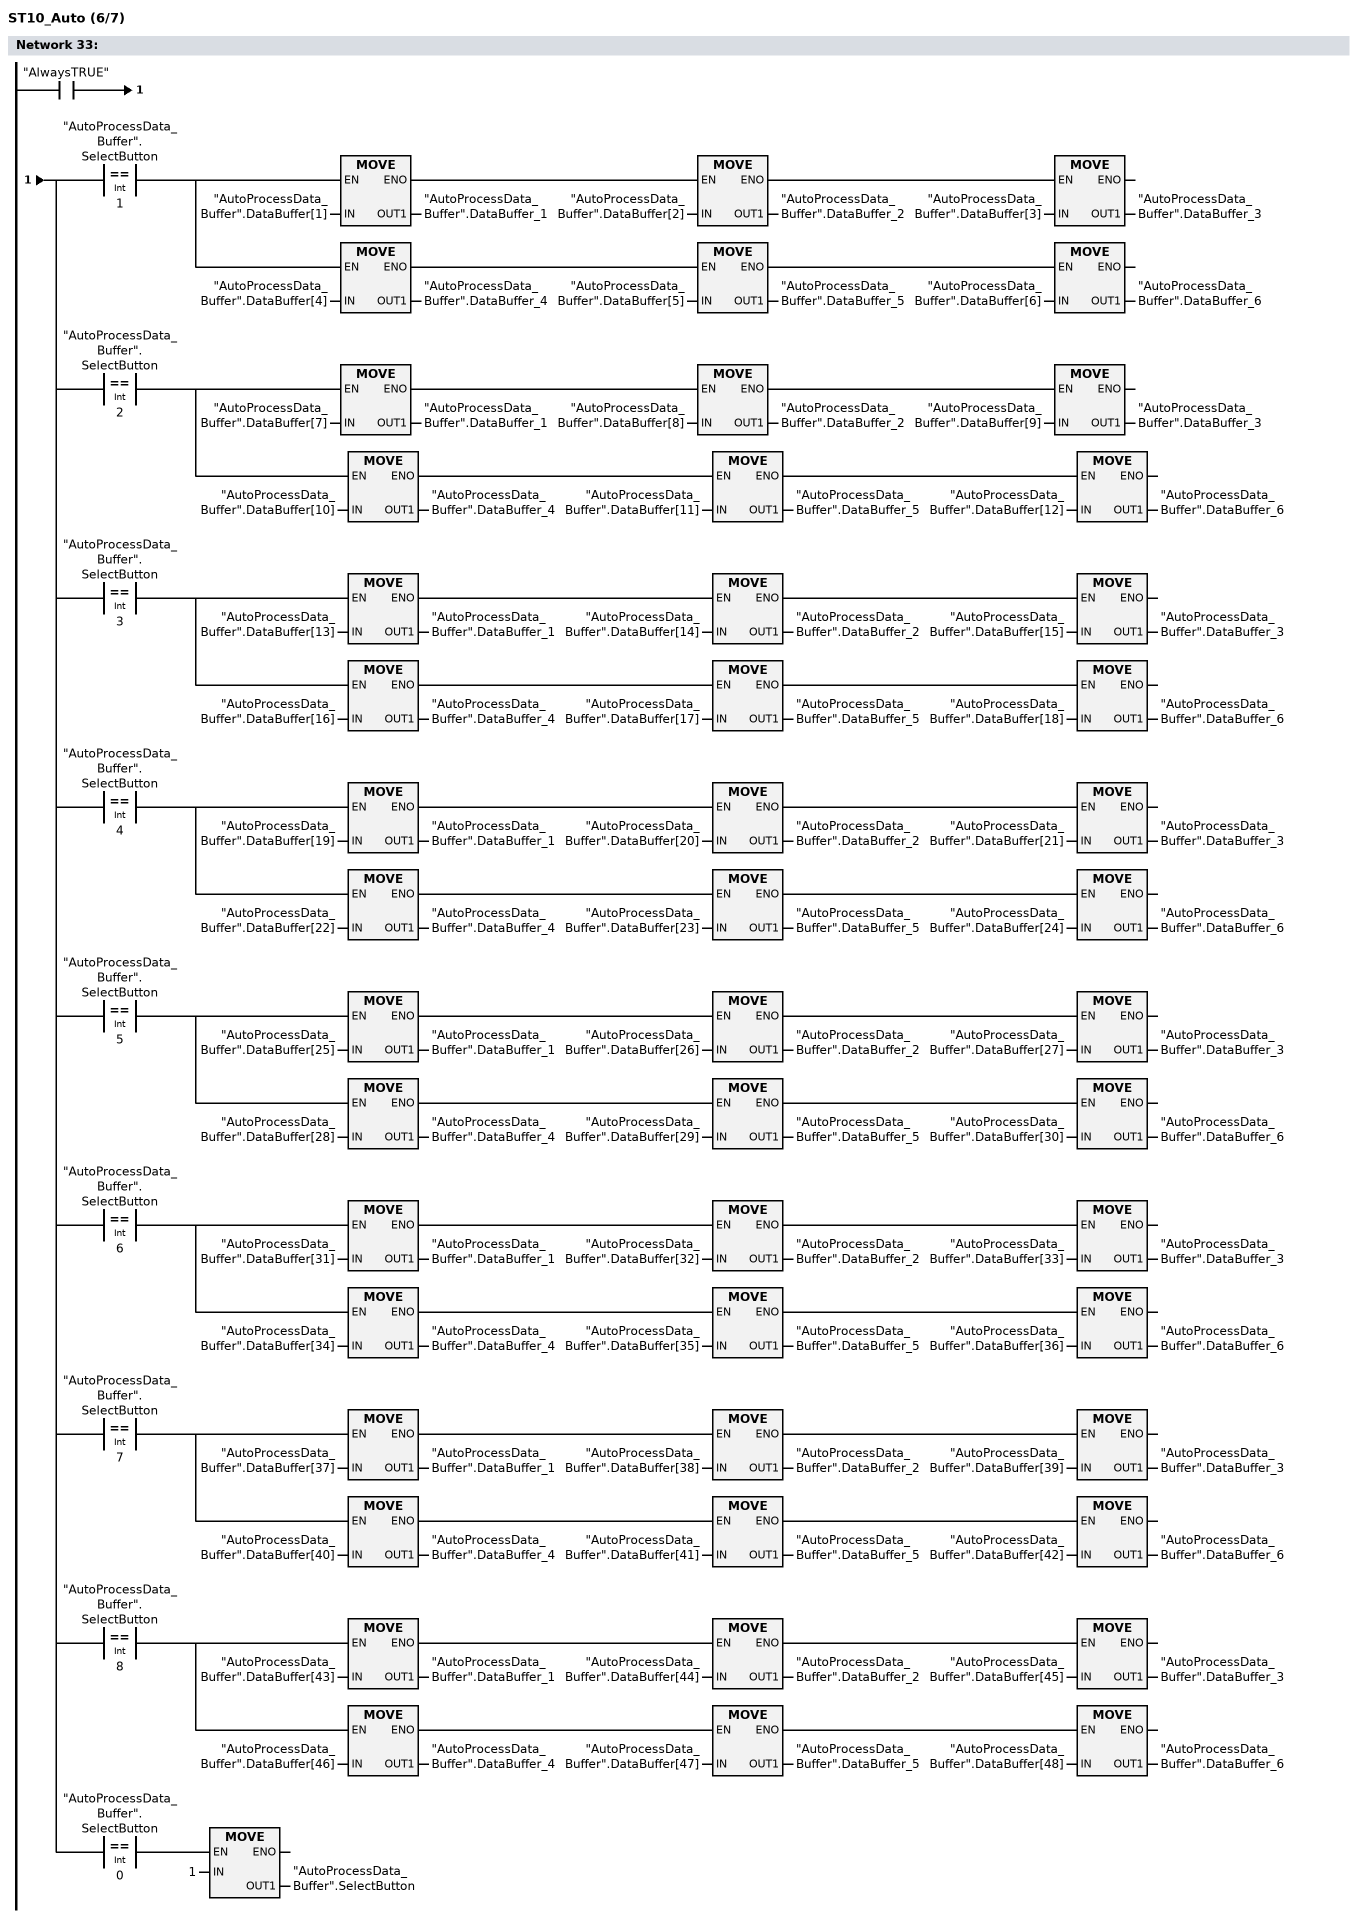
   RUNG wire#powerrail
      Contact( "AlwaysTRUE" )
      wire#w1
      { S7_Templates := "SrcType := Int" } EQ_Contact(in1 := "AutoProcessData_Buffer".SelectButton, in2 := 1)
      wire#w2
      Move(in := "AutoProcessData_Buffer".DataBuffer[1], out1 => "AutoProcessData_Buffer".DataBuffer_1)
      Move(in := "AutoProcessData_Buffer".DataBuffer[2], out1 => "AutoProcessData_Buffer".DataBuffer_2)
      Move(in := "AutoProcessData_Buffer".DataBuffer[3], out1 => "AutoProcessData_Buffer".DataBuffer_3)
   END_RUNG
   RUNG wire#w2
      Move(in := "AutoProcessData_Buffer".DataBuffer[4], out1 => "AutoProcessData_Buffer".DataBuffer_4)
      Move(in := "AutoProcessData_Buffer".DataBuffer[5], out1 => "AutoProcessData_Buffer".DataBuffer_5)
      Move(in := "AutoProcessData_Buffer".DataBuffer[6], out1 => "AutoProcessData_Buffer".DataBuffer_6)
   END_RUNG
   RUNG wire#w1
      { S7_Templates := "SrcType := Int" } EQ_Contact(in1 := "AutoProcessData_Buffer".SelectButton, in2 := 2)
      wire#w3
      Move(in := "AutoProcessData_Buffer".DataBuffer[7], out1 => "AutoProcessData_Buffer".DataBuffer_1)
      Move(in := "AutoProcessData_Buffer".DataBuffer[8], out1 => "AutoProcessData_Buffer".DataBuffer_2)
      Move(in := "AutoProcessData_Buffer".DataBuffer[9], out1 => "AutoProcessData_Buffer".DataBuffer_3)
   END_RUNG
   RUNG wire#w3
      Move(in := "AutoProcessData_Buffer".DataBuffer[10], out1 => "AutoProcessData_Buffer".DataBuffer_4)
      Move(in := "AutoProcessData_Buffer".DataBuffer[11], out1 => "AutoProcessData_Buffer".DataBuffer_5)
      Move(in := "AutoProcessData_Buffer".DataBuffer[12], out1 => "AutoProcessData_Buffer".DataBuffer_6)
   END_RUNG
   RUNG wire#w1
      { S7_Templates := "SrcType := Int" } EQ_Contact(in1 := "AutoProcessData_Buffer".SelectButton, in2 := 3)
      wire#w4
      Move(in := "AutoProcessData_Buffer".DataBuffer[13], out1 => "AutoProcessData_Buffer".DataBuffer_1)
      Move(in := "AutoProcessData_Buffer".DataBuffer[14], out1 => "AutoProcessData_Buffer".DataBuffer_2)
      Move(in := "AutoProcessData_Buffer".DataBuffer[15], out1 => "AutoProcessData_Buffer".DataBuffer_3)
   END_RUNG
   RUNG wire#w4
      Move(in := "AutoProcessData_Buffer".DataBuffer[16], out1 => "AutoProcessData_Buffer".DataBuffer_4)
      Move(in := "AutoProcessData_Buffer".DataBuffer[17], out1 => "AutoProcessData_Buffer".DataBuffer_5)
      Move(in := "AutoProcessData_Buffer".DataBuffer[18], out1 => "AutoProcessData_Buffer".DataBuffer_6)
   END_RUNG
   RUNG wire#w1
      { S7_Templates := "SrcType := Int" } EQ_Contact(in1 := "AutoProcessData_Buffer".SelectButton, in2 := 4)
      wire#w5
      Move(in := "AutoProcessData_Buffer".DataBuffer[19], out1 => "AutoProcessData_Buffer".DataBuffer_1)
      Move(in := "AutoProcessData_Buffer".DataBuffer[20], out1 => "AutoProcessData_Buffer".DataBuffer_2)
      Move(in := "AutoProcessData_Buffer".DataBuffer[21], out1 => "AutoProcessData_Buffer".DataBuffer_3)
   END_RUNG
   RUNG wire#w5
      Move(in := "AutoProcessData_Buffer".DataBuffer[22], out1 => "AutoProcessData_Buffer".DataBuffer_4)
      Move(in := "AutoProcessData_Buffer".DataBuffer[23], out1 => "AutoProcessData_Buffer".DataBuffer_5)
      Move(in := "AutoProcessData_Buffer".DataBuffer[24], out1 => "AutoProcessData_Buffer".DataBuffer_6)
   END_RUNG
   RUNG wire#w1
      { S7_Templates := "SrcType := Int" } EQ_Contact(in1 := "AutoProcessData_Buffer".SelectButton, in2 := 5)
      wire#w6
      Move(in := "AutoProcessData_Buffer".DataBuffer[25], out1 => "AutoProcessData_Buffer".DataBuffer_1)
      Move(in := "AutoProcessData_Buffer".DataBuffer[26], out1 => "AutoProcessData_Buffer".DataBuffer_2)
      Move(in := "AutoProcessData_Buffer".DataBuffer[27], out1 => "AutoProcessData_Buffer".DataBuffer_3)
   END_RUNG
   RUNG wire#w6
      Move(in := "AutoProcessData_Buffer".DataBuffer[28], out1 => "AutoProcessData_Buffer".DataBuffer_4)
      Move(in := "AutoProcessData_Buffer".DataBuffer[29], out1 => "AutoProcessData_Buffer".DataBuffer_5)
      Move(in := "AutoProcessData_Buffer".DataBuffer[30], out1 => "AutoProcessData_Buffer".DataBuffer_6)
   END_RUNG
   RUNG wire#w1
      { S7_Templates := "SrcType := Int" } EQ_Contact(in1 := "AutoProcessData_Buffer".SelectButton, in2 := 6)
      wire#w7
      Move(in := "AutoProcessData_Buffer".DataBuffer[31], out1 => "AutoProcessData_Buffer".DataBuffer_1)
      Move(in := "AutoProcessData_Buffer".DataBuffer[32], out1 => "AutoProcessData_Buffer".DataBuffer_2)
      Move(in := "AutoProcessData_Buffer".DataBuffer[33], out1 => "AutoProcessData_Buffer".DataBuffer_3)
   END_RUNG
   RUNG wire#w7
      Move(in := "AutoProcessData_Buffer".DataBuffer[34], out1 => "AutoProcessData_Buffer".DataBuffer_4)
      Move(in := "AutoProcessData_Buffer".DataBuffer[35], out1 => "AutoProcessData_Buffer".DataBuffer_5)
      Move(in := "AutoProcessData_Buffer".DataBuffer[36], out1 => "AutoProcessData_Buffer".DataBuffer_6)
   END_RUNG
   RUNG wire#w1
      { S7_Templates := "SrcType := Int" } EQ_Contact(in1 := "AutoProcessData_Buffer".SelectButton, in2 := 7)
      wire#w8
      Move(in := "AutoProcessData_Buffer".DataBuffer[37], out1 => "AutoProcessData_Buffer".DataBuffer_1)
      Move(in := "AutoProcessData_Buffer".DataBuffer[38], out1 => "AutoProcessData_Buffer".DataBuffer_2)
      Move(in := "AutoProcessData_Buffer".DataBuffer[39], out1 => "AutoProcessData_Buffer".DataBuffer_3)
   END_RUNG
   RUNG wire#w8
      Move(in := "AutoProcessData_Buffer".DataBuffer[40], out1 => "AutoProcessData_Buffer".DataBuffer_4)
      Move(in := "AutoProcessData_Buffer".DataBuffer[41], out1 => "AutoProcessData_Buffer".DataBuffer_5)
      Move(in := "AutoProcessData_Buffer".DataBuffer[42], out1 => "AutoProcessData_Buffer".DataBuffer_6)
   END_RUNG
   RUNG wire#w1
      { S7_Templates := "SrcType := Int" } EQ_Contact(in1 := "AutoProcessData_Buffer".SelectButton, in2 := 8)
      wire#w9
      Move(in := "AutoProcessData_Buffer".DataBuffer[43], out1 => "AutoProcessData_Buffer".DataBuffer_1)
      Move(in := "AutoProcessData_Buffer".DataBuffer[44], out1 => "AutoProcessData_Buffer".DataBuffer_2)
      Move(in := "AutoProcessData_Buffer".DataBuffer[45], out1 => "AutoProcessData_Buffer".DataBuffer_3)
   END_RUNG
   RUNG wire#w9
      Move(in := "AutoProcessData_Buffer".DataBuffer[46], out1 => "AutoProcessData_Buffer".DataBuffer_4)
      Move(in := "AutoProcessData_Buffer".DataBuffer[47], out1 => "AutoProcessData_Buffer".DataBuffer_5)
      Move(in := "AutoProcessData_Buffer".DataBuffer[48], out1 => "AutoProcessData_Buffer".DataBuffer_6)
   END_RUNG
   RUNG wire#w1
      { S7_Templates := "SrcType := Int" } EQ_Contact(in1 := "AutoProcessData_Buffer".SelectButton, in2 := 0)
      Move(in := 1, out1 => "AutoProcessData_Buffer".SelectButton)
   END_RUNG
   // the same network as SCL:
   IF "AlwaysTRUE" AND ("AutoProcessData_Buffer".SelectButton = 1) THEN
       "AutoProcessData_Buffer".DataBuffer_1 := "AutoProcessData_Buffer".DataBuffer[1];
       "AutoProcessData_Buffer".DataBuffer_2 := "AutoProcessData_Buffer".DataBuffer[2];
       "AutoProcessData_Buffer".DataBuffer_3 := "AutoProcessData_Buffer".DataBuffer[3];
       "AutoProcessData_Buffer".DataBuffer_4 := "AutoProcessData_Buffer".DataBuffer[4];
       "AutoProcessData_Buffer".DataBuffer_5 := "AutoProcessData_Buffer".DataBuffer[5];
       "AutoProcessData_Buffer".DataBuffer_6 := "AutoProcessData_Buffer".DataBuffer[6];
   END_IF;
   IF "AlwaysTRUE" AND ("AutoProcessData_Buffer".SelectButton = 2) THEN
       "AutoProcessData_Buffer".DataBuffer_1 := "AutoProcessData_Buffer".DataBuffer[7];
       "AutoProcessData_Buffer".DataBuffer_2 := "AutoProcessData_Buffer".DataBuffer[8];
       "AutoProcessData_Buffer".DataBuffer_3 := "AutoProcessData_Buffer".DataBuffer[9];
       "AutoProcessData_Buffer".DataBuffer_4 := "AutoProcessData_Buffer".DataBuffer[10];
       "AutoProcessData_Buffer".DataBuffer_5 := "AutoProcessData_Buffer".DataBuffer[11];
       "AutoProcessData_Buffer".DataBuffer_6 := "AutoProcessData_Buffer".DataBuffer[12];
   END_IF;
   IF "AlwaysTRUE" AND ("AutoProcessData_Buffer".SelectButton = 3) THEN
       "AutoProcessData_Buffer".DataBuffer_1 := "AutoProcessData_Buffer".DataBuffer[13];
       "AutoProcessData_Buffer".DataBuffer_2 := "AutoProcessData_Buffer".DataBuffer[14];
       "AutoProcessData_Buffer".DataBuffer_3 := "AutoProcessData_Buffer".DataBuffer[15];
       "AutoProcessData_Buffer".DataBuffer_4 := "AutoProcessData_Buffer".DataBuffer[16];
       "AutoProcessData_Buffer".DataBuffer_5 := "AutoProcessData_Buffer".DataBuffer[17];
       "AutoProcessData_Buffer".DataBuffer_6 := "AutoProcessData_Buffer".DataBuffer[18];
   END_IF;
   IF "AlwaysTRUE" AND ("AutoProcessData_Buffer".SelectButton = 4) THEN
       "AutoProcessData_Buffer".DataBuffer_1 := "AutoProcessData_Buffer".DataBuffer[19];
       "AutoProcessData_Buffer".DataBuffer_2 := "AutoProcessData_Buffer".DataBuffer[20];
       "AutoProcessData_Buffer".DataBuffer_3 := "AutoProcessData_Buffer".DataBuffer[21];
       "AutoProcessData_Buffer".DataBuffer_4 := "AutoProcessData_Buffer".DataBuffer[22];
       "AutoProcessData_Buffer".DataBuffer_5 := "AutoProcessData_Buffer".DataBuffer[23];
       "AutoProcessData_Buffer".DataBuffer_6 := "AutoProcessData_Buffer".DataBuffer[24];
   END_IF;
   IF "AlwaysTRUE" AND ("AutoProcessData_Buffer".SelectButton = 5) THEN
       "AutoProcessData_Buffer".DataBuffer_1 := "AutoProcessData_Buffer".DataBuffer[25];
       "AutoProcessData_Buffer".DataBuffer_2 := "AutoProcessData_Buffer".DataBuffer[26];
       "AutoProcessData_Buffer".DataBuffer_3 := "AutoProcessData_Buffer".DataBuffer[27];
       "AutoProcessData_Buffer".DataBuffer_4 := "AutoProcessData_Buffer".DataBuffer[28];
       "AutoProcessData_Buffer".DataBuffer_5 := "AutoProcessData_Buffer".DataBuffer[29];
       "AutoProcessData_Buffer".DataBuffer_6 := "AutoProcessData_Buffer".DataBuffer[30];
   END_IF;
   IF "AlwaysTRUE" AND ("AutoProcessData_Buffer".SelectButton = 6) THEN
       "AutoProcessData_Buffer".DataBuffer_1 := "AutoProcessData_Buffer".DataBuffer[31];
       "AutoProcessData_Buffer".DataBuffer_2 := "AutoProcessData_Buffer".DataBuffer[32];
       "AutoProcessData_Buffer".DataBuffer_3 := "AutoProcessData_Buffer".DataBuffer[33];
       "AutoProcessData_Buffer".DataBuffer_4 := "AutoProcessData_Buffer".DataBuffer[34];
       "AutoProcessData_Buffer".DataBuffer_5 := "AutoProcessData_Buffer".DataBuffer[35];
       "AutoProcessData_Buffer".DataBuffer_6 := "AutoProcessData_Buffer".DataBuffer[36];
   END_IF;
   IF "AlwaysTRUE" AND ("AutoProcessData_Buffer".SelectButton = 7) THEN
       "AutoProcessData_Buffer".DataBuffer_1 := "AutoProcessData_Buffer".DataBuffer[37];
       "AutoProcessData_Buffer".DataBuffer_2 := "AutoProcessData_Buffer".DataBuffer[38];
       "AutoProcessData_Buffer".DataBuffer_3 := "AutoProcessData_Buffer".DataBuffer[39];
       "AutoProcessData_Buffer".DataBuffer_4 := "AutoProcessData_Buffer".DataBuffer[40];
       "AutoProcessData_Buffer".DataBuffer_5 := "AutoProcessData_Buffer".DataBuffer[41];
       "AutoProcessData_Buffer".DataBuffer_6 := "AutoProcessData_Buffer".DataBuffer[42];
   END_IF;
   IF "AlwaysTRUE" AND ("AutoProcessData_Buffer".SelectButton = 8) THEN
       "AutoProcessData_Buffer".DataBuffer_1 := "AutoProcessData_Buffer".DataBuffer[43];
       "AutoProcessData_Buffer".DataBuffer_2 := "AutoProcessData_Buffer".DataBuffer[44];
       "AutoProcessData_Buffer".DataBuffer_3 := "AutoProcessData_Buffer".DataBuffer[45];
       "AutoProcessData_Buffer".DataBuffer_4 := "AutoProcessData_Buffer".DataBuffer[46];
       "AutoProcessData_Buffer".DataBuffer_5 := "AutoProcessData_Buffer".DataBuffer[47];
       "AutoProcessData_Buffer".DataBuffer_6 := "AutoProcessData_Buffer".DataBuffer[48];
   END_IF;
   IF "AlwaysTRUE" AND ("AutoProcessData_Buffer".SelectButton = 0) THEN
       "AutoProcessData_Buffer".SelectButton := 1;
   END_IF;
END_REGION

REGION Network 34
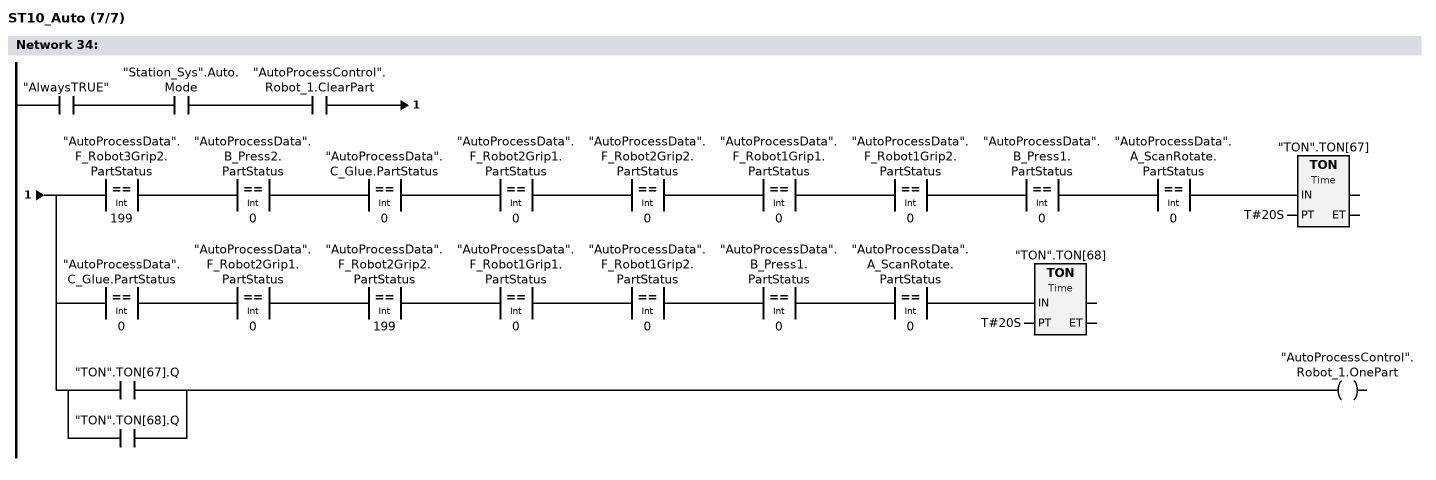
   RUNG wire#powerrail
      Contact( "AlwaysTRUE" )
      Contact( "Station_Sys".Auto.Mode )
      Contact( "AutoProcessControl".Robot_1.ClearPart )
      wire#w1
      { S7_Templates := "SrcType := Int" } EQ_Contact(in1 := "AutoProcessData".F_Robot3Grip2.PartStatus, in2 := 199)
      { S7_Templates := "SrcType := Int" } EQ_Contact(in1 := "AutoProcessData".B_Press2.PartStatus, in2 := 0)
      { S7_Templates := "SrcType := Int" } EQ_Contact(in1 := "AutoProcessData".C_Glue.PartStatus, in2 := 0)
      { S7_Templates := "SrcType := Int" } EQ_Contact(in1 := "AutoProcessData".F_Robot2Grip1.PartStatus, in2 := 0)
      { S7_Templates := "SrcType := Int" } EQ_Contact(in1 := "AutoProcessData".F_Robot2Grip2.PartStatus, in2 := 0)
      { S7_Templates := "SrcType := Int" } EQ_Contact(in1 := "AutoProcessData".F_Robot1Grip1.PartStatus, in2 := 0)
      { S7_Templates := "SrcType := Int" } EQ_Contact(in1 := "AutoProcessData".F_Robot1Grip2.PartStatus, in2 := 0)
      { S7_Templates := "SrcType := Int" } EQ_Contact(in1 := "AutoProcessData".B_Press1.PartStatus, in2 := 0)
      { S7_Templates := "SrcType := Int" } EQ_Contact(in1 := "AutoProcessData".A_ScanRotate.PartStatus, in2 := 0)
      { S7_Templates := "time_type := Time" } "TON".TON[67].TON(pt := T#20S, et =>)
   END_RUNG
   RUNG wire#w1
      { S7_Templates := "SrcType := Int" } EQ_Contact(in1 := "AutoProcessData".C_Glue.PartStatus, in2 := 0)
      { S7_Templates := "SrcType := Int" } EQ_Contact(in1 := "AutoProcessData".F_Robot2Grip1.PartStatus, in2 := 0)
      { S7_Templates := "SrcType := Int" } EQ_Contact(in1 := "AutoProcessData".F_Robot2Grip2.PartStatus, in2 := 199)
      { S7_Templates := "SrcType := Int" } EQ_Contact(in1 := "AutoProcessData".F_Robot1Grip1.PartStatus, in2 := 0)
      { S7_Templates := "SrcType := Int" } EQ_Contact(in1 := "AutoProcessData".F_Robot1Grip2.PartStatus, in2 := 0)
      { S7_Templates := "SrcType := Int" } EQ_Contact(in1 := "AutoProcessData".B_Press1.PartStatus, in2 := 0)
      { S7_Templates := "SrcType := Int" } EQ_Contact(in1 := "AutoProcessData".A_ScanRotate.PartStatus, in2 := 0)
      { S7_Templates := "time_type := Time" } "TON".TON[68].TON(pt := T#20S, et =>)
   END_RUNG
   RUNG wire#w1
      Contact( "TON".TON[67].Q )
      wire#w2
      Coil( "AutoProcessControl".Robot_1.OnePart )
   END_RUNG
   RUNG wire#w1
      Contact( "TON".TON[68].Q )
   END_RUNG wire#w2
   // the same network as SCL:
   #_w1 := "AlwaysTRUE" AND "Station_Sys".Auto.Mode AND "AutoProcessControl".Robot_1.ClearPart;
   "TON".TON[67].TON(IN := #_w1 AND ("AutoProcessData".F_Robot3Grip2.PartStatus = 199) AND ("AutoProcessData".B_Press2.PartStatus = 0) AND ("AutoProcessData".C_Glue.PartStatus = 0) AND ("AutoProcessData".F_Robot2Grip1.PartStatus = 0) AND ("AutoProcessData".F_Robot2Grip2.PartStatus = 0) AND ("AutoProcessData".F_Robot1Grip1.PartStatus = 0) AND ("AutoProcessData".F_Robot1Grip2.PartStatus = 0) AND ("AutoProcessData".B_Press1.PartStatus = 0) AND ("AutoProcessData".A_ScanRotate.PartStatus = 0),
                     PT := T#20S);
   "TON".TON[68].TON(IN := #_w1 AND ("AutoProcessData".C_Glue.PartStatus = 0) AND ("AutoProcessData".F_Robot2Grip1.PartStatus = 0) AND ("AutoProcessData".F_Robot2Grip2.PartStatus = 199) AND ("AutoProcessData".F_Robot1Grip1.PartStatus = 0) AND ("AutoProcessData".F_Robot1Grip2.PartStatus = 0) AND ("AutoProcessData".B_Press1.PartStatus = 0) AND ("AutoProcessData".A_ScanRotate.PartStatus = 0),
                     PT := T#20S);
   "AutoProcessControl".Robot_1.OnePart := #_w1 AND ("TON".TON[67].Q OR "TON".TON[68].Q);
END_REGION

REGION Network 36 (SCL)
   IF "Station_Sys".Initial.Running THEN
       FOR #FlankWord := 1 TO 99 DO
           "GeneralDebug".Debug[#FlankWord] := false;
       END_FOR;
   END_IF;
END_REGION
END_FUNCTION
